PROGRAM MAIN
VAR
	i : INT;
END_VAR

i := i + 1;

PRG_HA_SingleNode();	// call sample for UA_HistoryUpdate
PRG_HA_MultipleNodes();	// call sample for UA_HistoryUpdate with multiple nodes

END_PROGRAM

(* stored: Version 1.1.0.1, ProductVersion 3.1.4022.7
   POU MAIN: Id {3b66bfef-7a47-4837-bb7c-ec115028f14d}, SpecialFunc None *)
